(* IEC 61131-3 sources: pub-control-lib/test, 3 files *)

(* ---- CalcTest.st ---- *)
USING AxUnit;
USING Siemens.Calculator;

NAMESPACE Siemens.Calculator.Test

    {TestFixture}
    CLASS TestCalc

        VAR PROTECTED
            instAddCalc : Add;
            instSubCalc : Sub;
            values : Array[0..63] of REAL;
        END_VAR

        METHOD InitArray
            values[0] := REAL#3.0;
            values[1] := REAL#9.0;
            values[2] := REAL#30.0;
        END_METHOD

        {Test(operand1 := 9, operand2 := 30, result := 39)}
        {Test(operand1 := 9, operand2 := -30, result := -21)}
        METHOD PUBLIC TestAddCalc
            VAR_INPUT
                operand1 : REAL;
                operand2 : Real;
                result : Real;
            END_VAR
            VAR_TEMP
                myResult : REAL ;
            END_VAR
            myResult := instAddCalc.Calc(operand1, operand2);
            Assert.Equal(actual := myResult, expected := result);

        END_METHOD

        {Test(operand1 := 9, operand2 := 30, result := -21)}
        {Test(operand1 := 9, operand2 := -30, result := 39)}
        {Test(operand1 := 9, operand2 := 2, result := 7)}
        METHOD PUBLIC TestSubCalc
            VAR_INPUT
                operand1 : REAL;
                operand2 : Real;
                result : Real;
            END_VAR
            VAR_TEMP
                myResult : REAL ;
            END_VAR
            myResult := instSubCalc.Calc(operand1, operand2);
            Assert.Equal(actual := myResult, expected := result);

        END_METHOD

        {Test}
        METHOD PUBLIC TestAddArrayCalc
            VAR_TEMP
                myResult : Real;
            END_VAR
            THIS.InitArray();
            myResult := instAddCalc.ArrayCalc(values);
            Assert.Equal(actual := myResult, expected := 42);

        END_METHOD

        {Test}
        METHOD PUBLIC TestSubArrayCalc
            VAR_TEMP
                myResult : REAL;
            END_VAR
            THIS.InitArray();
            myResult := instSubCalc.ArrayCalc(values);
            Assert.Equal(actual := myResult, expected := -42);

        END_METHOD
    END_CLASS

END_NAMESPACE

(* ---- PubControlTankTest.st ---- *)
USING AxUnit;
USING Siemens.PubControl.TapBars;
USING Siemens.PubControl.Interfaces;
USING Siemens.PubControl.Types;

NAMESPACE Siemens.PubControl.Test

    {TestFixture}
    CLASS TestTank
        VAR
            tank : TankTap;
        END_VAR

        {FixtureSetup}
        METHOD PUBLIC ResetAndConfigTapBar
            VAR_TEMP
                result : BOOL;
            END_VAR

            tank.SetMaxLevel(UINT#900);

        END_METHOD

        {Test}
        METHOD PUBLIC TestLevel
            VAR_TEMP
                status : TankStatus;
                level : UINT := UINT#0;
            END_VAR
            tank.Tanking();
            level := tank.GetLevel();
            status := tank.GetStatus();
            Assert.Equal(expected := TankStatus#ACTIVE, actual := status);
            Assert.Equal(actual := level, expected := UINT#900);
        END_METHOD

        {Test(consume := REAL#2.0, exceptedlevel:= UINT#898)}
        METHOD PUBLIC Tapping
            VAR_INPUT
                consume : REAL;
                exceptedlevel : UINT := UINT#0;
            END_VAR
            VAR_TEMP
                status : TankStatus;
                currentlevel : UINT := UINT#0;
            END_VAR
            tank.Tanking();
            tank.Consume(consume);
            currentlevel := tank.GetLevel();
            status := tank.GetStatus();
            Assert.Equal(actual := status, expected := TankStatus#TAPPED);
            Assert.Equal(actual := currentlevel, expected := exceptedlevel);
        END_METHOD
    END_CLASS

END_NAMESPACE

(* ---- PubControlTapTest.st ---- *)
USING AxUnit;
USING Siemens.PubControl.TapBars;
USING Siemens.PubControl.Interfaces;

NAMESPACE Siemens.PubControl.Test

    {TestFixture}
    CLASS TestBasicTapBar

        VAR
            tapBar : BasicTapBar;
        END_VAR

        {FixtureSetup}
        METHOD PUBLIC ResetAndConfigTapBar
            VAR_TEMP
                result : BOOL;
            END_VAR

            tapBar.Reset();
            tapBar.WatchDogDiffTime := LTIME#60s;

        END_METHOD

        // {Test}
        // METHOD PUBLIC TestMeasure100ms
        //     VAR_TEMP
        //         flow : Real := REAL#0.0;
        //         consumption : Real := REAL#0.0;
        //     END_VAR
        //     //20 ml are 1 impulse
        //     tapBar.CalcImpulses(LTIME#100ms, 4, 5);
        //     consumption := tapBar.GetConsumption();
        //     flow := tapBar.GetFlow();
        //     Assert.InRange(consumption, 0.04, 0.002);
        //     Assert.Equal(actual := flow, expected := REAL#720.0);
        // END_METHOD
        // {Test}
        // METHOD PUBLIC SecondTestMeasure100ms
        //     VAR_TEMP
        //         flow : Real := REAL#0.0;
        //         consumption : Real := REAL#0.0;
        //     END_VAR
        //     //20 ml are 1 impulse
        //     tapBar.CalcImpulses(LTIME#100ms, 4, 5);
        //     consumption := tapBar.GetConsumption();
        //     flow := tapBar.GetFlow();
        //     Assert.Equal(actual := consumption, expected := REAL#0.04);
        //     Assert.Equal(actual := flow, expected := REAL#720.0);
        // END_METHOD
    END_CLASS

END_NAMESPACE
